// Mitsubishi GX Developer project: PLC_PCO520L2   PLC: Q06UDEH

PROGRAM AT_CART
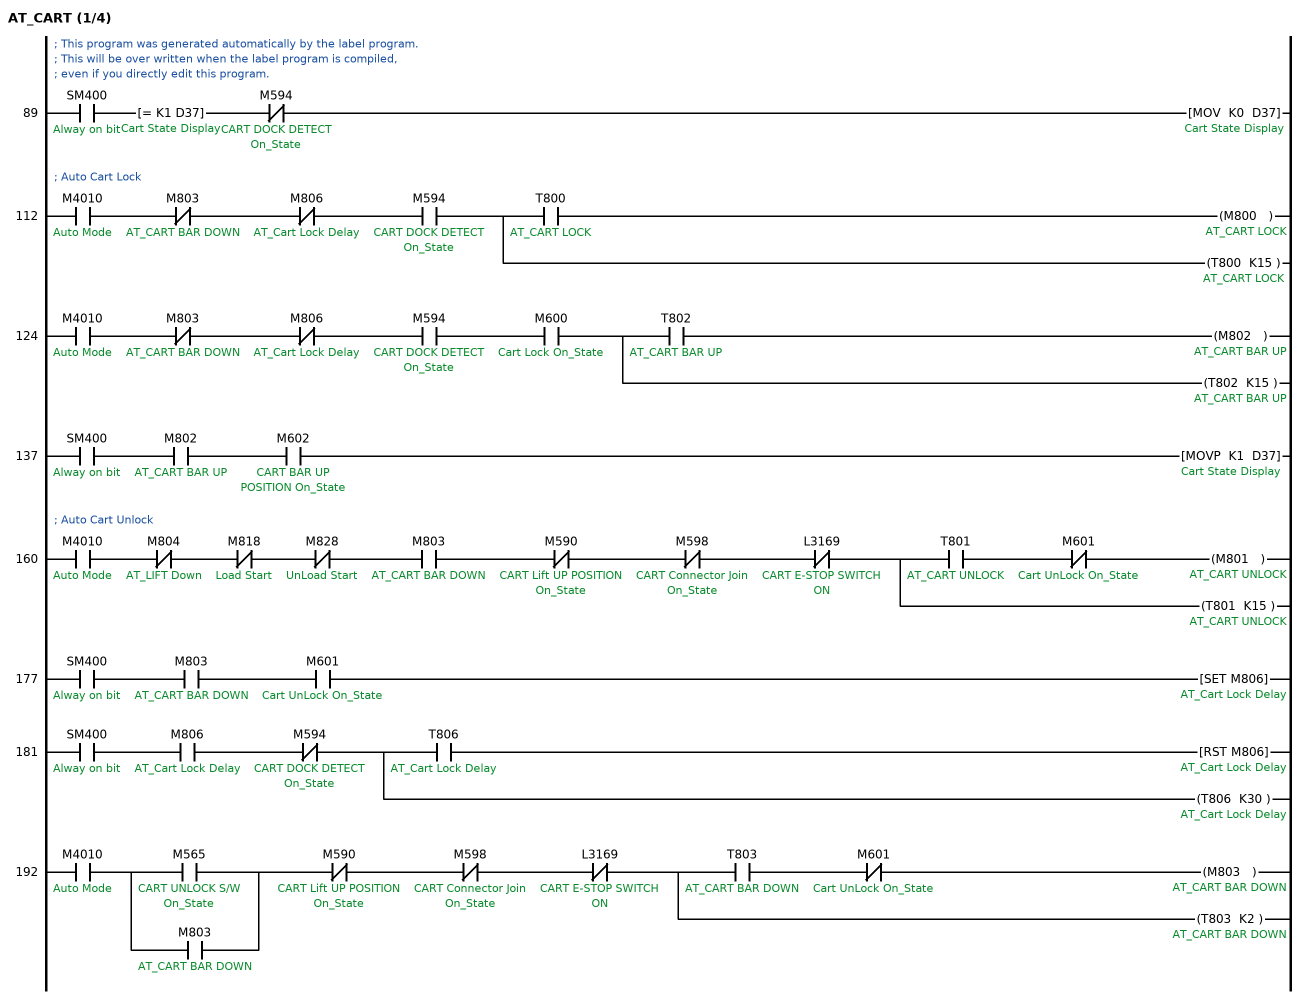
; This program was generated automatically by the label program.
; This will be over written when the label program is compiled,
; even if you directly edit this program.
89    LD      SM400  ; Alway on bit
      AND=    K1 D37  ; Cart State Display
      ANI     M594  ; CART DOCK DETECT On_State
      MOV     K0 D37
        [note] 0: Nothing
; Auto Cart Lock
112   LD      M4010  ; Auto Mode
      ANI     M803  ; AT_CART BAR DOWN
      ANI     M806  ; AT_Cart Lock Delay
      AND     M594  ; CART DOCK DETECT On_State
      MPS
      AND     T800  ; AT_CART LOCK
      OUT     M800  ; AT_CART LOCK
      MPP
      OUT     T800 K15  ; AT_CART LOCK
124   LD      M4010  ; Auto Mode
      ANI     M803  ; AT_CART BAR DOWN
      ANI     M806  ; AT_Cart Lock Delay
      AND     M594  ; CART DOCK DETECT On_State
      AND     M600  ; Cart Lock On_State
      MPS
      AND     T802  ; AT_CART BAR UP
      OUT     M802  ; AT_CART BAR UP
      MPP
      OUT     T802 K15  ; AT_CART BAR UP
137   LD      SM400  ; Alway on bit
      AND     M802  ; AT_CART BAR UP
      AND     M602  ; CART BAR UP POSITION On_State
      MOVP    K1 D37
        [note] 1: CART IDLE
; Auto Cart Unlock
160   LD      M4010  ; Auto Mode
      ANI     M804  ; AT_LIFT Down
      ANI     M818  ; Load Start
      ANI     M828  ; UnLoad Start
      AND     M803  ; AT_CART BAR DOWN
      ANI     M590  ; CART Lift UP POSITION On_State
      ANI     M598  ; CART Connector Join On_State
      ANI     L3169  ; CART E-STOP SWITCH ON
      MPS
      AND     T801  ; AT_CART UNLOCK
      ANI     M601  ; Cart UnLock On_State
      OUT     M801  ; AT_CART UNLOCK
      MPP
      OUT     T801 K15  ; AT_CART UNLOCK
177   LD      SM400  ; Alway on bit
      AND     M803  ; AT_CART BAR DOWN
      AND     M601  ; Cart UnLock On_State
      SET     M806  ; AT_Cart Lock Delay
181   LD      SM400  ; Alway on bit
      AND     M806  ; AT_Cart Lock Delay
      ANI     M594  ; CART DOCK DETECT On_State
      MPS
      AND     T806  ; AT_Cart Lock Delay
      RST     M806  ; AT_Cart Lock Delay
      MPP
      OUT     T806 K30  ; AT_Cart Lock Delay
192   LD      M4010  ; Auto Mode
      LD      M565  ; CART UNLOCK S/W On_State
      OR      M803  ; AT_CART BAR DOWN
      ANB
      ANI     M590  ; CART Lift UP POSITION On_State
      ANI     M598  ; CART Connector Join On_State
      ANI     L3169  ; CART E-STOP SWITCH ON
      MPS
      AND     T803  ; AT_CART BAR DOWN
      ANI     M601  ; Cart UnLock On_State
      OUT     M803  ; AT_CART BAR DOWN
      MPP
      OUT     T803 K2  ; AT_CART BAR DOWN
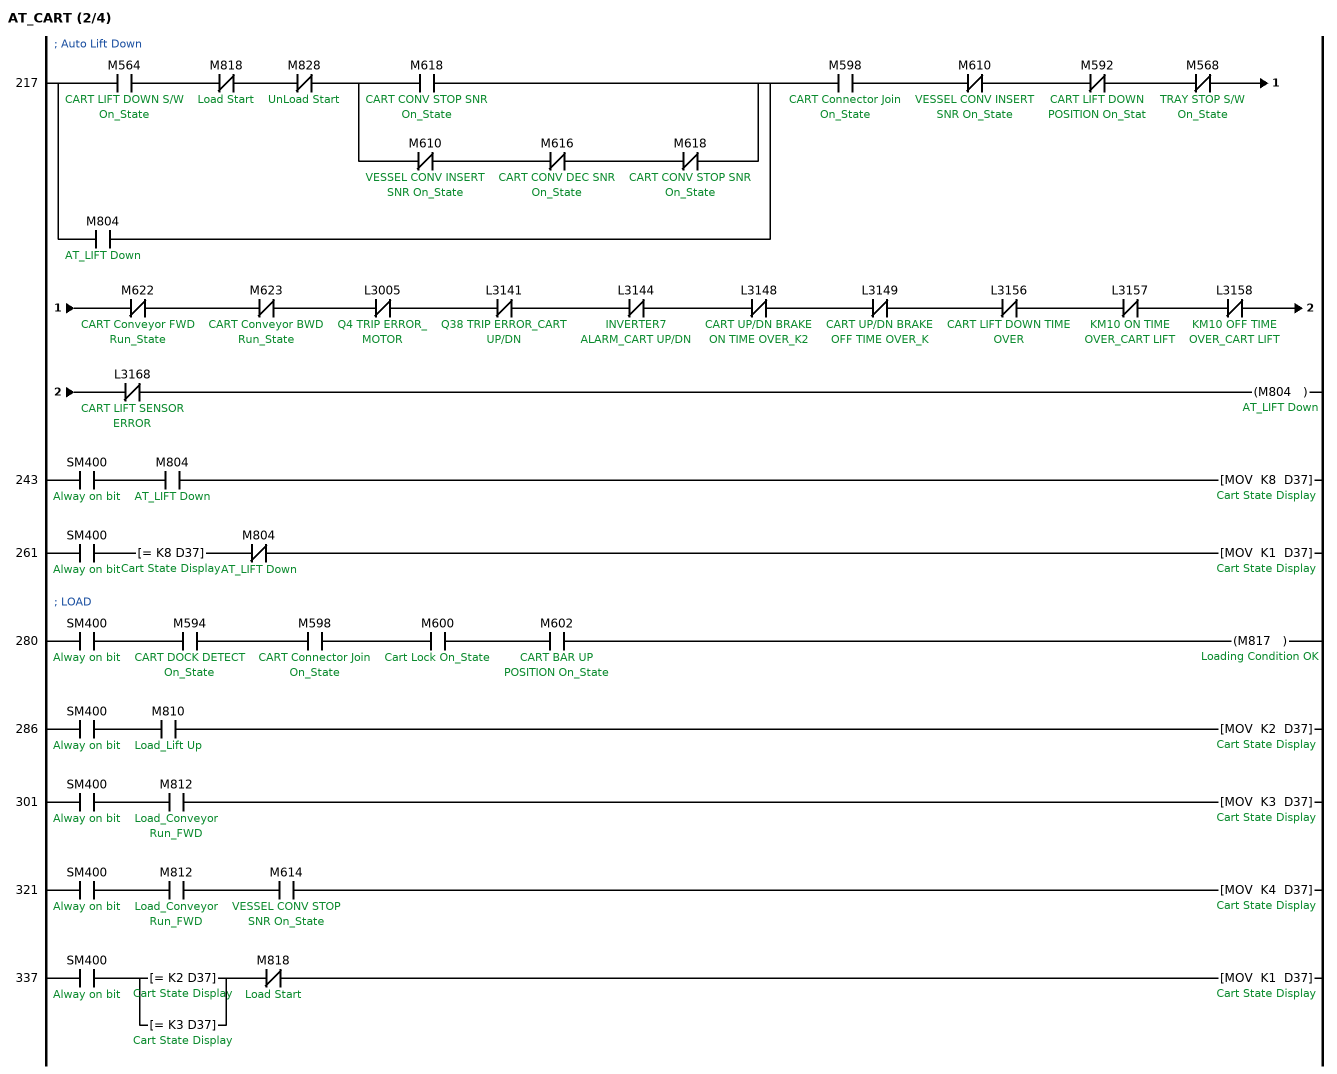
; Auto Lift Down
217   LD      M564  ; CART LIFT DOWN S/W On_State
      ANI     M818  ; Load Start
      ANI     M828  ; UnLoad Start
      LD      M618  ; CART CONV STOP SNR On_State
      LDI     M610  ; VESSEL CONV INSERT SNR On_State
      ANI     M616  ; CART CONV DEC SNR On_State
      ANI     M618  ; CART CONV STOP SNR On_State
      ORB
      ANB
      OR      M804  ; AT_LIFT Down
      AND     M598  ; CART Connector Join On_State
      ANI     M610  ; VESSEL CONV INSERT SNR On_State
      ANI     M592  ; CART LIFT DOWN  POSITION On_Stat
      ANI     M568  ; TRAY STOP S/W On_State
      ANI     M622  ; CART Conveyor FWD Run_State
      ANI     M623  ; CART Conveyor BWD Run_State
      ANI     L3005  ; Q4 TRIP ERROR_MOTOR
      ANI     L3141  ; Q38 TRIP ERROR_CART UP/DN
      ANI     L3144  ; INVERTER7 ALARM_CART UP/DN
      ANI     L3148  ; CART UP/DN BRAKE ON TIME OVER_K2
      ANI     L3149  ; CART UP/DN BRAKE OFF TIME OVER_K
      ANI     L3156  ; CART LIFT DOWN TIME OVER
      ANI     L3157  ; KM10 ON TIME OVER_CART LIFT
      ANI     L3158  ; KM10 OFF TIME OVER_CART LIFT
      ANI     L3168  ; CART LIFT SENSOR ERROR
      OUT     M804  ; AT_LIFT Down
243   LD      SM400  ; Alway on bit
      AND     M804  ; AT_LIFT Down
      MOV     K8 D37
        [note] 8:Lift Down in progress
261   LD      SM400  ; Alway on bit
      AND=    K8 D37  ; Cart State Display
      ANI     M804  ; AT_LIFT Down
      MOV     K1 D37
        [note] 1:Cart Idle
; LOAD
280   LD      SM400  ; Alway on bit
      AND     M594  ; CART DOCK DETECT On_State
      AND     M598  ; CART Connector Join On_State
      AND     M600  ; Cart Lock On_State
      AND     M602  ; CART BAR UP POSITION On_State
      OUT     M817  ; Loading Condition OK
286   LD      SM400  ; Alway on bit
      AND     M810  ; Load_Lift Up
      MOV     K2 D37
        [note] 2:Loading-Lift UP
301   LD      SM400  ; Alway on bit
      AND     M812  ; Load_Conveyor Run_FWD
      MOV     K3 D37
        [note] 3: Loading-Conveyor Running
321   LD      SM400  ; Alway on bit
      AND     M812  ; Load_Conveyor Run_FWD
      AND     M614  ; VESSEL CONV STOP SNR On_State
      MOV     K4 D37
        [note] 4: Load Completed
337   LD      SM400  ; Alway on bit
      LD=     K2 D37  ; Cart State Display
      OR=     K3 D37  ; Cart State Display
      ANB
      ANI     M818  ; Load Start
      MOV     K1 D37
        [note] 1: Cart Idle
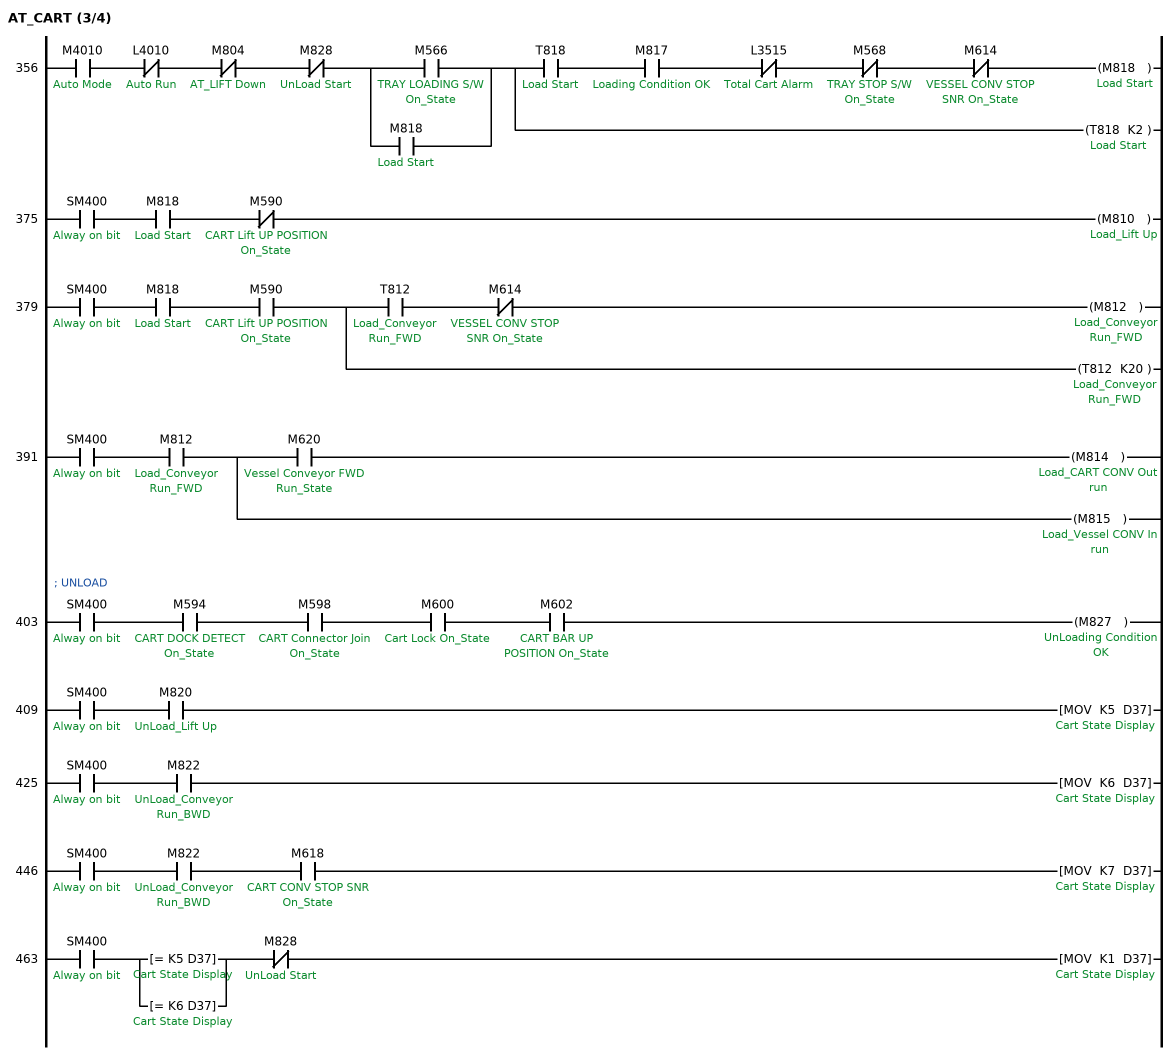
356   LD      M4010  ; Auto Mode
      ANI     L4010  ; Auto Run
      ANI     M804  ; AT_LIFT Down
      ANI     M828  ; UnLoad Start
      LD      M566  ; TRAY LOADING S/W On_State
      OR      M818  ; Load Start
      ANB
      MPS
      AND     T818  ; Load Start
      AND     M817  ; Loading Condition OK
      ANI     L3515  ; Total Cart Alarm
      ANI     M568  ; TRAY STOP S/W On_State
      ANI     M614  ; VESSEL CONV STOP SNR On_State
      OUT     M818  ; Load Start
      MPP
      OUT     T818 K2  ; Load Start
375   LD      SM400  ; Alway on bit
      AND     M818  ; Load Start
      ANI     M590  ; CART Lift UP POSITION On_State
      OUT     M810  ; Load_Lift Up
379   LD      SM400  ; Alway on bit
      AND     M818  ; Load Start
      AND     M590  ; CART Lift UP POSITION On_State
      MPS
      AND     T812  ; Load_Conveyor Run_FWD
      ANI     M614  ; VESSEL CONV STOP SNR On_State
      OUT     M812  ; Load_Conveyor Run_FWD
      MPP
      OUT     T812 K20  ; Load_Conveyor Run_FWD
391   LD      SM400  ; Alway on bit
      AND     M812  ; Load_Conveyor Run_FWD
      MPS
      AND     M620  ; Vessel Conveyor FWD Run_State
      OUT     M814  ; Load_CART CONV Out run
      MPP
      OUT     M815  ; Load_Vessel CONV In run
; UNLOAD
403   LD      SM400  ; Alway on bit
      AND     M594  ; CART DOCK DETECT On_State
      AND     M598  ; CART Connector Join On_State
      AND     M600  ; Cart Lock On_State
      AND     M602  ; CART BAR UP POSITION On_State
      OUT     M827  ; UnLoading Condition OK
409   LD      SM400  ; Alway on bit
      AND     M820  ; UnLoad_Lift Up
      MOV     K5 D37
        [note] 5:UnLoading-Lift UP
425   LD      SM400  ; Alway on bit
      AND     M822  ; UnLoad_Conveyor Run_BWD
      MOV     K6 D37
        [note] 6: UnLoading-Conveyor Running
446   LD      SM400  ; Alway on bit
      AND     M822  ; UnLoad_Conveyor Run_BWD
      AND     M618  ; CART CONV STOP SNR On_State
      MOV     K7 D37
        [note] 7: UnLoad Completed
463   LD      SM400  ; Alway on bit
      LD=     K5 D37  ; Cart State Display
      OR=     K6 D37  ; Cart State Display
      ANB
      ANI     M828  ; UnLoad Start
      MOV     K1 D37
        [note] 1: Cart Idle
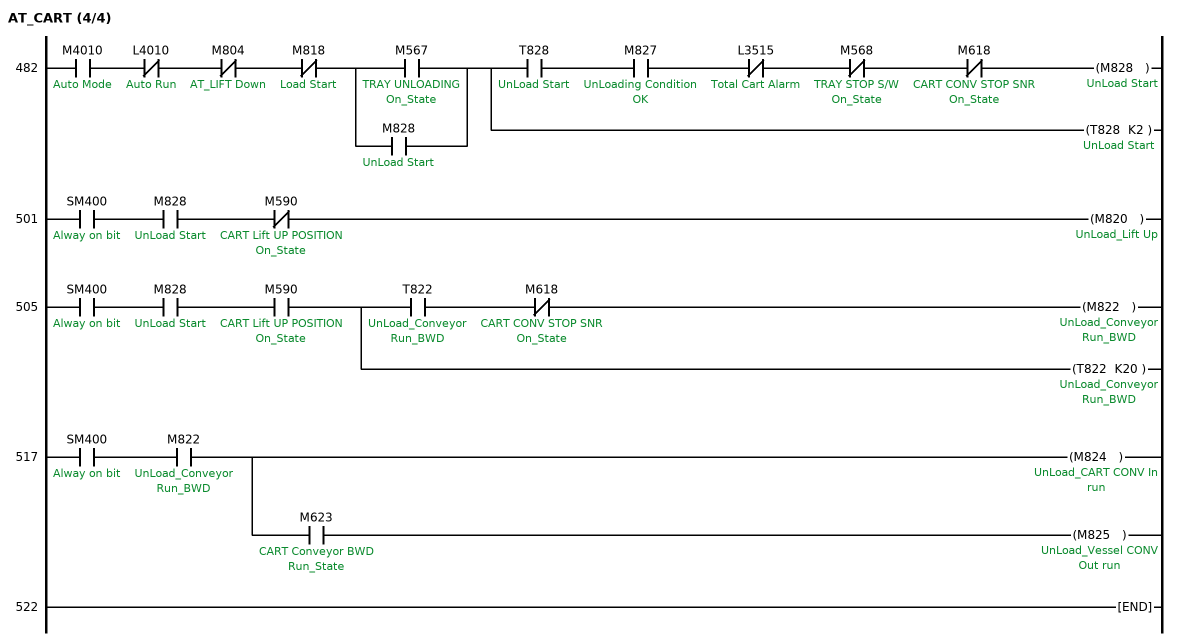
482   LD      M4010  ; Auto Mode
      ANI     L4010  ; Auto Run
      ANI     M804  ; AT_LIFT Down
      ANI     M818  ; Load Start
      LD      M567  ; TRAY UNLOADING On_State
      OR      M828  ; UnLoad Start
      ANB
      MPS
      AND     T828  ; UnLoad Start
      AND     M827  ; UnLoading Condition OK
      ANI     L3515  ; Total Cart Alarm
      ANI     M568  ; TRAY STOP S/W On_State
      ANI     M618  ; CART CONV STOP SNR On_State
      OUT     M828  ; UnLoad Start
      MPP
      OUT     T828 K2  ; UnLoad Start
501   LD      SM400  ; Alway on bit
      AND     M828  ; UnLoad Start
      ANI     M590  ; CART Lift UP POSITION On_State
      OUT     M820  ; UnLoad_Lift Up
505   LD      SM400  ; Alway on bit
      AND     M828  ; UnLoad Start
      AND     M590  ; CART Lift UP POSITION On_State
      MPS
      AND     T822  ; UnLoad_Conveyor Run_BWD
      ANI     M618  ; CART CONV STOP SNR On_State
      OUT     M822  ; UnLoad_Conveyor Run_BWD
      MPP
      OUT     T822 K20  ; UnLoad_Conveyor Run_BWD
517   LD      SM400  ; Alway on bit
      AND     M822  ; UnLoad_Conveyor Run_BWD
      OUT     M824  ; UnLoad_CART CONV In run
      AND     M623  ; CART Conveyor BWD Run_State
      OUT     M825  ; UnLoad_Vessel CONV Out run
522   END
END_PROGRAM
